TYPE TFMachineTransportIN :
STRUCT
	Mode : Mode;
	PowerOk : BOOL;
	SensorAir : BOOL;
	Sensor24Volt : BOOL;
END_STRUCT
END_TYPE

(* stored: Version 1.1.0.1, ProductVersion 3.1.4024.11
   DUT TFMachineTransportIN: Id {0c4f8951-f7a9-44e1-a807-fec028b79fee} *)
